KUKA KRL program: style1pick1opt1AutoRR.src, style1pick1opt1AutoRR.dat

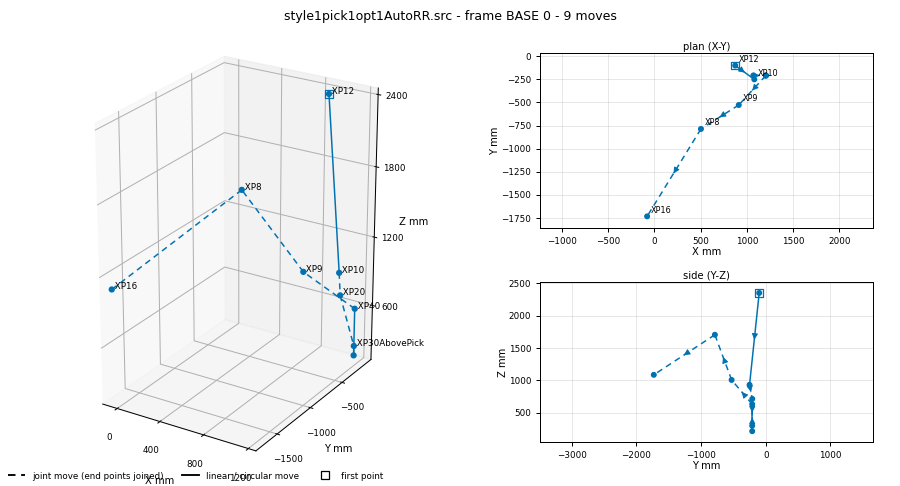
[picture p0: tool path of style1pick1opt1AutoRR.src in frame BASE 0, 9 of 9 moves have a stored position in this frame; points joined in program order, loops and branches not executed]
--- style1pick1opt1AutoRR.src ---
&ACCESS RVO1
&REL 61
&COMMENT 03-10-R1 RED RABBIT PICK
&PARAM EDITMASK = *
&PARAM DISKPATH = KRC:\R1\Program\StylePicks\Options
DEF style1pick1opt1AutoRR( )
   ;FOLD INI
      ;FOLD BASISTECH INI
         GLOBAL INTERRUPT DECL 3 WHEN $STOPMESS==TRUE DO IR_STOPM ( )
         INTERRUPT ON 3
         BAS (#INITMOV,0 )
      ;ENDFOLD (BASISTECH INI)
      ;FOLD USER INI
         ;Make your modifications here

      ;ENDFOLD (USER INI)
   ;ENDFOLD (INI)
;********************************
; Gestamp Standards
; Line - BMW G65 (cell 03)
; Robot 03-10-R1 (BMW-03-10-R1-MH1)
; Application - RED RABBIT PICK AT PICKUP 1 (STATION 1) WITH EOAT 1
;********************************
;NOTE: CALLED BY Style1Opt10AutoRR (OPTION 12, RED RABBIT); SAME PATH AS style1pick1opt1 PLUS P16
;NOTE: IT STARTS A NUT PRELOAD (NUT_START AT P12) ALTHOUGH NO WELDING FOLLOWS (F14)
;NOTE: THE WAIT FOR STATEMENTS BELOW HAVE NO TIMEOUT AND NO MESSAGE (F15)
;PICKUP 1 REQUEST - AC_pickUPCheck(1): WAIT SIGNAL $IN[65] di065PickupMachine1 ON,
;THEN SIGNALS $OUT[65] do065PickupClear1 OFF, $OUT[23] do023PickClearTooling OFF
   ;FOLD PickUp[1] Request
      ;FOLD ;%{h}
         ;Params IlfProvider=ac_zoneilf; AC_CmdZones=PickUp; AC_CmdParam=1; AC_ZoneRepo=False; AC_Blending=False
      ;ENDFOLD
      AC_pickUPCheck (1)
   ;ENDFOLD
;WAIT GRIPPER EMPTY BEFORE ANY GRIPPER COMMAND - SIGNALS $IN[253] di253PartPresent1 OFF,
;$IN[254] di254PartPresent2 OFF (GESTAMP REVIEW POINT 14)
;FOLD WAIT FOR ( NOT IN 253 'di253PartPresent1' ) AND ( NOT IN 254 'di254PartPresent2' );%{PE}%R 8.3.43,%MKUKATPBASIS,%CEXT_WAIT_FOR,%VEXT_WAIT_FOR,%P 2:, 4:NOT, 5:$IN, 6:253, 7:di253PartPresent1, 9:AND, 10:, 12:NOT, 13:$IN, 14:254, 15:di254PartPresent2, 17:
WAIT FOR  (  NOT $IN[253] ) AND (  NOT $IN[254])
;ENDFOLD
;GRIPPER 1 OPEN - SIGNALS $OUT[249] do249Group1Home ON, $OUT[250] do250Group1Work OFF, WAIT 0.2 S,
;THEN CHECK $IN[257] di257Cylinder1Home ON, $IN[258] di258Cylinder1Work OFF (STRATEGY 1)
;NOTE: THE HIDDEN FORM PARAMETERS NOW MATCH THE CALL (WERE setgripper=4;setstate=2, F31)
   ;FOLD Gripper SET [1]Gripper1 State=[1]OPEN Wait 0.2[s] Check with Strategy 1 ;%{PE}
      ;FOLD Parameters Parameters ;%{h}
         ;Params IlfProvider=GripperTech.GripperSet;setgripper=1;setstate=1;setcont=nocont;waittime=0.2;errorstrategy=1
      ;ENDFOLD
      GRPg_SetStateAndCheck(1, 1, 0.2, 1)
   ;ENDFOLD

;APPROACH PICKUP - P12
;THEN P10, P20, P30AbovePick (ABOVE THE PART), AtPick3 (PICK POSITION)
;NUT 1 - TRIGGER ON THE MOTION TO P12 (DISTANCE = 0: FIRES WHEN THE MOTION STARTS): NUT_START=TRUE
;STARTS THE NUT PRELOAD (PRELOAD, CALLED FROM sps.sub) FOR THE FIRST NUT
;NOTE: THE TRIGGER STANDS BEFORE THE INLINE FORM, SO A TOUCH UP CANNOT DELETE IT; IT ACTS ON
;NOTE: THE NEXT MOTION. A BLOCK SELECTION ONTO THE MOTION FOLD SKIPS IT (SELECT THE TRIGGER
;NOTE: LINE): NO NUT 1 PRELOAD IS REQUESTED (F14)
;NOTE: NUT_START IS SET ALSO IN DRY CYCLE AND WHEN STEPPING IN T1/T2 (F04, F11)
TRIGGER WHEN DISTANCE = 0 DELAY = 0 DO NUT_START=TRUE
;FOLD PTP P12 Vel=100 % PDAT15 Tool[1]:TOOL 1 Base[0];%{PE}%R 8.3.43,%MKUKATPBASIS,%CMOVE,%VPTP,%P 1:PTP, 2:P12, 3:, 5:100, 7:PDAT15
$BWDSTART=FALSE
PDAT_ACT=PPDAT15
FDAT_ACT=FP12
BAS(#PTP_PARAMS,100)
PTP XP12
;ENDFOLD
;FOLD LIN P10 CONT Vel=2 m/s CPDAT5 Tool[1]:TOOL 1 Base[0];%{PE}%R 8.3.43,%MKUKATPBASIS,%CMOVE,%VLIN,%P 1:LIN, 2:P10, 3:C_DIS C_DIS, 5:2, 7:CPDAT5
$BWDSTART=FALSE
LDAT_ACT=LCPDAT5
FDAT_ACT=FP10
BAS(#CP_PARAMS,2)
LIN XP10 C_DIS C_DIS
;ENDFOLD
   ;FOLD PTP P20 CONT Vel=100 % PDAT2 Tool[1]:TOOL 1 Base[0];%{PE}%R 8.3.43,%MKUKATPBASIS,%CMOVE,%VPTP,%P 1:PTP, 2:P20, 3:C_DIS, 5:100, 7:PDAT2
      $BWDSTART=FALSE
      PDAT_ACT=PPDAT2
      FDAT_ACT=FP20
      BAS(#PTP_PARAMS,100)
      PTP XP20 C_DIS
   ;ENDFOLD
   ;FOLD PTP P30AbovePick CONT Vel=100 % PDAT4 Tool[1]:TOOL 1 Base[0];%{PE}%R 8.3.43,%MKUKATPBASIS,%CMOVE,%VPTP,%P 1:PTP, 2:P30AbovePick, 3:C_DIS, 5:100, 7:PDAT4
      $BWDSTART=FALSE
      PDAT_ACT=PPDAT4
      FDAT_ACT=FP30AbovePick
      BAS(#PTP_PARAMS,100)
      PTP XP30AbovePick C_DIS
   ;ENDFOLD
;NOTE: THE FOLD TITLE SAYS AtPick1; THE FORM DATA AND THE CODE MOVE TO AtPick3
   ;FOLD LIN AtPick1 Vel=2 m/s CPDAT1 Tool[1]:TOOL 1 Base[0];%{PE}%R 8.3.43,%MKUKATPBASIS,%CMOVE,%VLIN,%P 1:LIN, 2:AtPick3, 3:, 5:2, 7:CPDAT1
      $BWDSTART=FALSE
      LDAT_ACT=LCPDAT1
      FDAT_ACT=FAtPick3
      BAS(#CP_PARAMS,2)
      LIN XAtPick3
   ;ENDFOLD

;GRIPPER 1 CLOSE - SIGNALS $OUT[249] do249Group1Home OFF, $OUT[250] do250Group1Work ON, WAIT 0.2 S,
;THEN CHECK $IN[257] di257Cylinder1Home OFF, $IN[258] di258Cylinder1Work ON (STRATEGY 1)
;NOTE: THE HIDDEN FORM PARAMETERS NOW MATCH THE CALL (WERE setgripper=4;setstate=2, F31)
   ;FOLD Gripper SET [1]Gripper1 State=[2]CLOSE Wait 0.2[s] Check with Strategy 1 ;%{PE}
      ;FOLD Parameters Parameters ;%{h}
         ;Params IlfProvider=GripperTech.GripperSet;setgripper=1;setstate=2;setcont=nocont;waittime=0.2;errorstrategy=1
      ;ENDFOLD
      GRPg_SetStateAndCheck(1, 2, 0.2, 1)
   ;ENDFOLD

;OUTSIDE DRY CYCLE ONLY (SIGNAL $IN[4] di004UseDryCycle OFF): PART-PRESENT WAIT AND
;$OUT[18] do018Part1InGripper
;NOTE: $IN[4] IS RE-READ HERE AND AT EVERY LATER STEP OF THE CYCLE, NOT LATCHED (F05)
IF NOT di004UseDryCycle THEN
;WAIT PART IN GRIPPER - SIGNALS $IN[253] di253PartPresent1 ON, $IN[254] di254PartPresent2 ON
;FOLD WAIT FOR ( IN 253 'di253PartPresent1' ) AND ( IN 254 'di254PartPresent2' );%{PE}%R 8.3.43,%MKUKATPBASIS,%CEXT_WAIT_FOR,%VEXT_WAIT_FOR,%P 2:, 4:, 5:$IN, 6:253, 7:di253PartPresent1, 9:AND, 10:, 12:, 13:$IN, 14:254, 15:di254PartPresent2, 17:
WAIT FOR  ( $IN[253] ) AND ( $IN[254] )
;ENDFOLD
;PART IN GRIPPER - SIGNAL $OUT[18] do018Part1InGripper ON
;NOTE: THE FORM TEXT do018PartInGripper1 IS NOT A DECLARED NAME (DECLARED: do018Part1InGripper).
;NOTE: $OUT[18] IS SET HERE AND RESET AT THE DROP - IT DOES NOT FOLLOW THE SENSORS (GESTAMP POINT 9)
   ;FOLD OUT 18 'do018PartInGripper1' State=TRUE ;%{PE}%R 8.3.43,%MKUKATPBASIS,%COUT,%VOUTX,%P 2:18, 3:do018PartInGripper1, 5:TRUE, 6:
      $OUT[18]=TRUE
   ;ENDFOLD
ENDIF

;LEAVE PICKUP 1 - P40 (ABOVE AtPick3), P9, P8, P16 (60 %)
   ;FOLD LIN P40 Vel=2 m/s CPDAT2 Tool[1]:TOOL 1 Base[0];%{PE}%R 8.3.43,%MKUKATPBASIS,%CMOVE,%VLIN,%P 1:LIN, 2:P40, 3:, 5:2, 7:CPDAT2
      $BWDSTART=FALSE
      LDAT_ACT=LCPDAT2
      FDAT_ACT=FP40
      BAS(#CP_PARAMS,2)
      LIN XP40
   ;ENDFOLD
;FOLD PTP P9 Vel=100 % PDAT13 Tool[1]:TOOL 1 Base[0];%{PE}%R 8.3.43,%MKUKATPBASIS,%CMOVE,%VPTP,%P 1:PTP, 2:P9, 3:, 5:100, 7:PDAT13
$BWDSTART=FALSE
PDAT_ACT=PPDAT13
FDAT_ACT=FP9
BAS(#PTP_PARAMS,100)
PTP XP9
;ENDFOLD
;FOLD PTP P8 Vel=100 % PDAT12 Tool[1]:TOOL 1 Base[0];%{PE}%R 8.3.43,%MKUKATPBASIS,%CMOVE,%VPTP,%P 1:PTP, 2:P8, 3:, 5:100, 7:PDAT12
$BWDSTART=FALSE
PDAT_ACT=PPDAT12
FDAT_ACT=FP8
BAS(#PTP_PARAMS,100)
PTP XP8
;ENDFOLD

;FOLD PTP P16 Vel=60 % PDAT18 Tool[1]:TOOL 1 Base[0];%{PE}%R 8.3.43,%MKUKATPBASIS,%CMOVE,%VPTP,%P 1:PTP, 2:P16, 3:, 5:60, 7:PDAT18
$BWDSTART=FALSE
PDAT_ACT=PPDAT18
FDAT_ACT=FP16
BAS(#PTP_PARAMS,60)
PTP XP16
;ENDFOLD
;PICKUP 1 CLEAR - AC_pickUP(1,TRUE): SIGNAL $OUT[65] do065PickupClear1 ON
   ;FOLD PickUp[1] Reset
      ;FOLD ;%{h}
         ;Params IlfProvider=ac_zoneilf; AC_CmdZones=PickUp; AC_CmdParam=1; AC_ZoneRepo=True; AC_Blending=False
      ;ENDFOLD
      AC_pickUP (1,True)
   ;ENDFOLD
END

--- style1pick1opt1AutoRR.dat ---
&ACCESS RVO1
&REL 61
&COMMENT St1_PICK_GE4
&PARAM EDITMASK = *
&PARAM DISKPATH = KRC:\R1\Program\StylePicks\Options
DEFDAT  style1pick1opt1AutoRR
;FOLD EXTERNAL DECLARATIONS;%{PE}%MKUKATPBASIS,%CEXT,%VCOMMON,%P
;FOLD BASISTECH EXT;%{PE}%MKUKATPBASIS,%CEXT,%VEXT,%P
EXT  BAS (BAS_COMMAND  :IN,REAL  :IN )
DECL INT SUCCESS
;ENDFOLD (BASISTECH EXT)
;FOLD USER EXT;%{E}%MKUKATPUSER,%CEXT,%VEXT,%P
;Make here your modifications

;ENDFOLD (USER EXT)
;ENDFOLD (EXTERNAL DECLARATIONS)
DECL E6POS XTag4={X -612.686,Y -1589.39600,Z 2916.51807,A 84.5120,B -104.062,C 7.85700,S 2,T 2,E1 0.0,E2 0.0,E3 0.0,E4 0.0,E5 0.0,E6 0.0}
DECL FDAT FTag4={TOOL_NO 7,BASE_NO 0,IPO_FRAME #BASE}
DECL PDAT PPDAT1={VEL 100.000,ACC 100.000,APO_DIST 1000.00,APO_MODE #CDIS,GEAR_JERK 50.0000,EXAX_IGN 0}
DECL E6POS XTag3={X -570.159,Y -2455.64600,Z 462.298,A 90.7960,B -176.000,C -0.0550000,S 2,T 2,E1 0.0,E2 0.0,E3 0.0,E4 0.0,E5 0.0,E6 0.0}
DECL FDAT FTag3={TOOL_NO 7,BASE_NO 0,IPO_FRAME #BASE}
DECL PDAT PPDAT2={VEL 100.000,ACC 100.000,APO_DIST 500.000,APO_MODE #CDIS,GEAR_JERK 50.0000,EXAX_IGN 0}
DECL E6POS XTag1={X -570.159,Y -2469.59692,Z 262.786,A 90.7960,B -176.000,C -0.0560000,S 2,T 2,E1 0.0,E2 0.0,E3 0.0,E4 0.0,E5 0.0,E6 0.0}
DECL FDAT FTag1={TOOL_NO 7,BASE_NO 0,IPO_FRAME #BASE}
DECL LDAT LCPDAT1={VEL 2.00000,ACC 100.000,APO_DIST 0.0,APO_FAC 50.0000,AXIS_VEL 100.000,AXIS_ACC 100.000,ORI_TYP #VAR,CIRC_TYP #BASE,JERK_FAC 50.0000,GEAR_JERK 50.0000,EXAX_IGN 0}
DECL E6POS XTag2={X -570.159,Y -2466.10889,Z 312.664,A 90.7960,B -176.000,C -0.0560000,S 2,T 2,E1 0.0,E2 0.0,E3 0.0,E4 0.0,E5 0.0,E6 0.0}
DECL FDAT FTag2={TOOL_NO 7,BASE_NO 0,IPO_FRAME #BASE}
DECL LDAT LCPDAT2={VEL 2.00000,ACC 100.000,APO_DIST 100.000,APO_FAC 50.0000,AXIS_VEL 100.000,AXIS_ACC 100.000,ORI_TYP #VAR,CIRC_TYP #BASE,JERK_FAC 50.0000,GEAR_JERK 50.0000,EXAX_IGN 0}
DECL BASIS_SUGG_T LAST_BASIS={POINT1[] "P0                      ",POINT2[] "P0                      ",CP_PARAMS[] "CPDAT0                  ",PTP_PARAMS[] "PDAT0                   ",CONT[] "                        ",CP_VEL[] "2.0                     ",PTP_VEL[] " 100                    ",SYNC_PARAMS[] "SYNCDAT                 ",SPL_NAME[] "S0                      ",A_PARAMS[] "ADAT0                   "}
DECL E6POS XP20={X 1070.46545,Y -208.124084,Z 714.012268,A -91.4409,B -0.232809603,C 0.168291062,S 2,T 3,E1 0.0,E2 0.0,E3 0.0,E4 0.0,E5 0.0,E6 0.0}
DECL FDAT FP20={TOOL_NO 1,BASE_NO 0,IPO_FRAME #BASE,POINT2[] " ",TQ_STATE FALSE}
DECL E6POS XP10={X 1081.09485,Y -250.197342,Z 931.476,A -96.8303,B 37.9899406,C -15.7576666,S 2,T 3,E1 0.0,E2 0.0,E3 0.0,E4 0.0,E5 0.0,E6 0.0}
DECL FDAT FP10={TOOL_NO 1,BASE_NO 0,IPO_FRAME #BASE,POINT2[] " ",TQ_STATE FALSE}
DECL E6POS XP30={X -602.469604,Y -2473.76245,Z 446.371094,A -89.4232254,B -2.67896390,C -179.996689,S 2,T 2,E1 0.0,E2 0.0,E3 0.0,E4 0.0,E5 0.0,E6 0.0}
DECL FDAT FP30={TOOL_NO 7,BASE_NO 0,IPO_FRAME #BASE,POINT2[] " ",TQ_STATE FALSE}
DECL E6POS XAtPick3={X 1206.28552,Y -208.912048,Z 214.158249,A -91.4409,B -0.232809141,C 0.168289974,S 2,T 3,E1 0.0,E2 0.0,E3 0.0,E4 0.0,E5 0.0,E6 0.0}
DECL FDAT FAtPick3={TOOL_NO 1,BASE_NO 0,IPO_FRAME #BASE,POINT2[] " ",TQ_STATE FALSE}
DECL E6POS XP1={X -603.354553,Y -2477.18481,Z 667.120239,A -89.3294754,B 0.653617203,C -179.853607,S 2,T 10,E1 0.0,E2 0.0,E3 0.0,E4 0.0,E5 0.0,E6 0.0}
DECL FDAT FP1={TOOL_NO 7,BASE_NO 0,IPO_FRAME #BASE,POINT2[] " ",TQ_STATE FALSE}
DECL LDAT LCPDAT3={VEL 2.00000,ACC 100.000,APO_DIST 100.000,APO_FAC 50.0000,AXIS_VEL 100.000,AXIS_ACC 100.000,ORI_TYP #VAR,CIRC_TYP #BASE,JERK_FAC 50.0000,GEAR_JERK 50.0000,EXAX_IGN 0}
DECL E6POS XP40={X 1206.28552,Y -208.912048,Z 630.625366,A -91.4409,B -0.232809082,C 0.168290034,S 2,T 3,E1 0.0,E2 0.0,E3 0.0,E4 0.0,E5 0.0,E6 0.0}
DECL FDAT FP40={TOOL_NO 1,BASE_NO 0,IPO_FRAME #BASE,POINT2[] " ",TQ_STATE FALSE}
DECL E6POS XP50={X 1206.28552,Y -208.912048,Z 409.521729,A -91.4413757,B -0.232714087,C 0.168696448,S 2,T 3,E1 0.0,E2 0.0,E3 0.0,E4 0.0,E5 0.0,E6 0.0}
DECL FDAT FP50={TOOL_NO 1,BASE_NO 0,IPO_FRAME #BASE,POINT2[] " ",TQ_STATE FALSE}
DECL E6POS XP60={X 671.407898,Y -378.268097,Z 2030.44653,A -89.8029327,B 7.84505653,C 24.4156590,S 2,T 3,E1 0.0,E2 0.0,E3 0.0,E4 0.0,E5 0.0,E6 0.0}
DECL FDAT FP60={TOOL_NO 1,BASE_NO 0,IPO_FRAME #BASE,POINT2[] " ",TQ_STATE FALSE}
DECL PDAT PPDAT3={VEL 100.000,ACC 100.000,APO_DIST 100.000,APO_MODE #CDIS,GEAR_JERK 50.0000,EXAX_IGN 0}
DECL PDAT PPDAT4={VEL 100.000,ACC 100.000,APO_DIST 10.0000,APO_MODE #CDIS,GEAR_JERK 50.0000,EXAX_IGN 0}
DECL E6POS XP70={X 1525.90320,Y -261.054626,Z 1246.12451,A 16.2779942,B 28.5338478,C 22.5772171,S 2,T 42,E1 0.0,E2 0.0,E3 0.0,E4 0.0,E5 0.0,E6 0.0}
DECL FDAT FP70={TOOL_NO 1,BASE_NO 0,IPO_FRAME #BASE,POINT2[] " ",TQ_STATE FALSE}
DECL PDAT PPDAT5={VEL 100.000,ACC 100.000,APO_DIST 500.000,APO_MODE #CDIS,GEAR_JERK 50.0000,EXAX_IGN 0}
DECL E6POS XP30ABOVEPICK={X 1206.28552,Y -208.912048,Z 298.869263,A -91.4409,B -0.232809111,C 0.168290,S 2,T 3,E1 0.0,E2 0.0,E3 0.0,E4 0.0,E5 0.0,E6 0.0}
DECL FDAT FP30AbovePick={TOOL_NO 1,BASE_NO 0,IPO_FRAME #BASE,POINT2[] " ",TQ_STATE FALSE}
DECL E6POS XP2={X -599.756165,Y -2478.73,Z 369.150330,A -89.4027710,B -3.84103417,C 179.935089,S 2,T 2,E1 0.0,E2 0.0,E3 0.0,E4 0.0,E5 0.0,E6 0.0}
DECL FDAT FP2={TOOL_NO 7,BASE_NO 0,IPO_FRAME #BASE,POINT2[] " ",TQ_STATE FALSE}
DECL PDAT PPDAT6={VEL 100.000,ACC 100.000,APO_DIST 100.000,GEAR_JERK 50.0000,EXAX_IGN 0}
DECL E6POS XP3={X -599.698364,Y -2469.82422,Z 501.779144,A -89.4027710,B -3.84103417,C 179.935089,S 2,T 2,E1 0.0,E2 0.0,E3 0.0,E4 0.0,E5 0.0,E6 0.0}
DECL FDAT FP3={TOOL_NO 7,BASE_NO 0,IPO_FRAME #BASE,POINT2[] " ",TQ_STATE FALSE}
DECL PDAT PPDAT7={VEL 100.000,ACC 100.000,APO_DIST 100.000,GEAR_JERK 50.0000,EXAX_IGN 0}
DECL PDAT PPDAT0={VEL 100.000,ACC 100.000,APO_DIST 1000.00,APO_MODE #CDIS,GEAR_JERK 50.0000,EXAX_IGN 0}
DECL E6POS XP0={X 1206.28552,Y -208.912048,Z 573.307922,A -91.4409,B -0.232809082,C 0.168290049,S 2,T 3,E1 0.0,E2 0.0,E3 0.0,E4 0.0,E5 0.0,E6 0.0}
DECL FDAT FP0={TOOL_NO 1,BASE_NO 0,IPO_FRAME #BASE,POINT2[] " ",TQ_STATE FALSE}
DECL LDAT LCPDAT4={VEL 2.00000,ACC 100.000,APO_DIST 100.000,APO_FAC 50.0000,AXIS_VEL 100.000,AXIS_ACC 100.000,ORI_TYP #VAR,CIRC_TYP #BASE,JERK_FAC 50.0000,GEAR_JERK 50.0000,EXAX_IGN 0}
DECL PDAT PPDAT8={VEL 100.000,ACC 100.000,APO_DIST 1000.00,APO_MODE #CDIS,GEAR_JERK 50.0000,EXAX_IGN 0}
DECL E6POS XP4={X 0.0,Y 0.0,Z 0.0,A 0.0,B 0.0,C 0.0,S 2,T 3,E1 0.0,E2 0.0,E3 0.0,E4 0.0,E5 0.0,E6 0.0}
DECL FDAT FP4={TOOL_NO 0,BASE_NO 0,IPO_FRAME #BASE,POINT2[] " ",TQ_STATE FALSE}
DECL PDAT PPDAT9={VEL 100.000,ACC 100.000,APO_DIST 1000.00,APO_MODE #CDIS,GEAR_JERK 50.0000,EXAX_IGN 0}
DECL E6POS XP5={X 1206.28552,Y -208.912048,Z 1092.82214,A -91.4409,B -0.232809037,C 0.168290079,S 2,T 3,E1 0.0,E2 0.0,E3 0.0,E4 0.0,E5 0.0,E6 0.0}
DECL FDAT FP5={TOOL_NO 1,BASE_NO 0,IPO_FRAME #BASE,POINT2[] " ",TQ_STATE FALSE}
DECL E6POS XP6={X 12.7359648,Y -130.494156,Z 3309.79932,A -58.5948639,B -68.7112122,C 63.6888771,S 3,T 2,E1 0.0,E2 0.0,E3 0.0,E4 0.0,E5 0.0,E6 0.0}
DECL FDAT FP6={TOOL_NO 1,BASE_NO 0,IPO_FRAME #BASE,POINT2[] " ",TQ_STATE FALSE}
DECL PDAT PPDAT10={VEL 100.000,ACC 100.000,APO_DIST 100.000,APO_MODE #CDIS,GEAR_JERK 50.0000,EXAX_IGN 0}
DECL E6POS XP7={X -1067.77161,Y -2105.70923,Z -1670.46326,A -142.262650,B 26.2927914,C -143.375824,S 2,T 2,E1 0.0,E2 0.0,E3 0.0,E4 0.0,E5 0.0,E6 0.0}
DECL FDAT FP7={TOOL_NO 1,BASE_NO 3,IPO_FRAME #TCP,POINT2[] " ",TQ_STATE FALSE}
DECL PDAT PPDAT11={VEL 100.000,ACC 100.000,APO_DIST 100.000,APO_MODE #CDIS,GEAR_JERK 50.0000,EXAX_IGN 0}
DECL E6POS XP8={X 504.083313,Y -786.363220,Z 1705.62256,A -111.705475,B 40.2604485,C 19.4570847,S 2,T 2,E1 0.0,E2 0.0,E3 0.0,E4 0.0,E5 0.0,E6 0.0}
DECL FDAT FP8={TOOL_NO 1,BASE_NO 0,IPO_FRAME #BASE,POINT2[] " ",TQ_STATE FALSE}
DECL PDAT PPDAT12={VEL 100.000,ACC 100.000,APO_DIST 100.000,APO_MODE #CDIS,GEAR_JERK 50.0000,EXAX_IGN 0}
DECL LDAT LCPDAT5={VEL 2.00000,ACC 100.000,APO_DIST 100.000,APO_FAC 50.0000,AXIS_VEL 100.000,AXIS_ACC 100.000,ORI_TYP #VAR,CIRC_TYP #BASE,JERK_FAC 50.0000,GEAR_JERK 50.0000,EXAX_IGN 0}
DECL E6POS XP9={X 913.201294,Y -527.473816,Z 1006.97571,A -91.4454117,B -0.232742429,C 0.168951720,S 2,T 3,E1 0.0,E2 0.0,E3 0.0,E4 0.0,E5 0.0,E6 0.0}
DECL FDAT FP9={TOOL_NO 1,BASE_NO 0,IPO_FRAME #BASE,POINT2[] " ",TQ_STATE FALSE}
DECL PDAT PPDAT13={VEL 100.000,ACC 100.000,APO_DIST 100.000,APO_MODE #CDIS,GEAR_JERK 50.0000,EXAX_IGN 0}
DECL E6POS XP11={X 874.811584,Y -100.693855,Z 2352.82324,A -4.40713501,B 2.42977476,C 0.669138968,S 2,T 10,E1 0.0,E2 0.0,E3 0.0,E4 0.0,E5 0.0,E6 0.0}
DECL FDAT FP11={TOOL_NO 1,BASE_NO 0,IPO_FRAME #BASE,POINT2[] " ",TQ_STATE FALSE}
DECL PDAT PPDAT14={VEL 100.000,ACC 100.000,APO_DIST 100.000,APO_MODE #CDIS,GEAR_JERK 50.0000,EXAX_IGN 0}
DECL E6POS XP12={X 874.811584,Y -100.693466,Z 2352.82349,A -4.40710449,B 2.42972946,C 0.669244647,S 2,T 10,E1 0.0,E2 0.0,E3 0.0,E4 0.0,E5 0.0,E6 0.0}
DECL FDAT FP12={TOOL_NO 1,BASE_NO 0,IPO_FRAME #BASE,POINT2[] " ",TQ_STATE FALSE}
DECL PDAT PPDAT15={VEL 100.000,ACC 100.000,APO_DIST 100.000,APO_MODE #CDIS,GEAR_JERK 50.0000,EXAX_IGN 0}
DECL E6POS XP13={X 257.073029,Y -1149.13025,Z 1934.72095,A -130.412979,B 3.09674358,C 77.3307953,S 2,T 2,E1 0.0,E2 0.0,E3 0.0,E4 0.0,E5 0.0,E6 0.0}
DECL FDAT FP13={TOOL_NO 1,BASE_NO 0,IPO_FRAME #BASE,POINT2[] " ",TQ_STATE FALSE}
DECL PDAT PPDAT16={VEL 100.000,ACC 100.000,APO_DIST 100.000,APO_MODE #CDIS,GEAR_JERK 50.0000,EXAX_IGN 0}
DECL PDAT PPDAT17={VEL 100.000,ACC 100.000,APO_DIST 100.000,APO_MODE #CDIS,GEAR_JERK 50.0000,EXAX_IGN 0}
DECL E6POS XP14={X -3704.29346,Y 1.10223198,Z -449.805786,A -178.368118,B 0.266879767,C 179.968445,S 2,T 34,E1 0.0,E2 0.0,E3 0.0,E4 0.0,E5 0.0,E6 0.0}
DECL FDAT FP14={TOOL_NO 1,BASE_NO 3,IPO_FRAME #TCP,POINT2[] " ",TQ_STATE FALSE}
DECL LDAT LCPDAT0={VEL 2.00000,ACC 100.000,APO_DIST 100.000,APO_FAC 50.0000,AXIS_VEL 100.000,AXIS_ACC 100.000,ORI_TYP #VAR,CIRC_TYP #BASE,JERK_FAC 50.0000,GEAR_JERK 50.0000,EXAX_IGN 0}
DECL E6POS XP15={X -3704.29346,Y 1.10223198,Z -449.805786,A -178.368118,B 0.266879767,C 179.968445,S 2,T 34,E1 0.0,E2 0.0,E3 0.0,E4 0.0,E5 0.0,E6 0.0}
DECL FDAT FP15={TOOL_NO 1,BASE_NO 3,IPO_FRAME #TCP,POINT2[] " ",TQ_STATE FALSE}
DECL PDAT PPDAT18={VEL 100.000,ACC 100.000,APO_DIST 100.000,APO_MODE #CDIS,GEAR_JERK 50.0000,EXAX_IGN 0}
DECL E6POS XP16={X -77.5694046,Y -1731.18909,Z 1086.30457,A -91.6320343,B 0.265882939,C -0.0392194763,S 2,T 34,E1 0.0,E2 0.0,E3 0.0,E4 0.0,E5 0.0,E6 0.0}
DECL FDAT FP16={TOOL_NO 1,BASE_NO 0,IPO_FRAME #BASE,POINT2[] " ",TQ_STATE FALSE}
ENDDAT
